SUBAPPLICATION Uebung_026_sub (* Spiegelabfolge (6) *)
  (* Standard: 61499-2 *)
  (* Version 1.0, 2024-02-05, franz *)
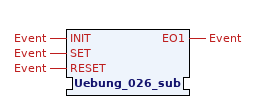
  EVENT_INPUT
    INIT;
    SET;
    RESET;
  END_EVENT
  EVENT_OUTPUT
    EO1;
  END_EVENT
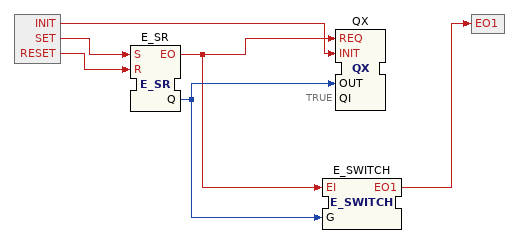
  FBS
    E_SR : E_SR;
    QX : QX(QI := TRUE);
    E_SWITCH : E_SWITCH;
  END_FBS
  EVENT_CONNECTIONS
    E_SR.EO TO QX.REQ;
    E_SR.EO TO E_SWITCH.EI;
    SET TO E_SR.S;
    RESET TO E_SR.R;
    INIT TO QX.INIT;
    E_SWITCH.EO1 TO EO1;
  END_CONNECTIONS
  DATA_CONNECTIONS
    E_SR.Q TO QX.OUT;
    E_SR.Q TO E_SWITCH.G;
  END_CONNECTIONS
END_SUBAPPLICATION
